Staubli VAL3: GeometryRS.dtx

public bool bIsScara = true
public bool bLinear = true
public bool bUseUserCenter
public bool bUseUserLimit = true
public num nSyncDist = 1
public num nWinDownStream
public num nWinUpStream
pointRs pVision[3]
  [0] = {x=319.933347, y=-456.969728, z=-77.119399, rx=-180, ry=0, rz=-52.793717, shoulder=lefty, fatherId=world[0]}
  [1] = {x=263.701989, y=-456.674668, z=-77.415466, rx=-180, ry=0, rz=-52.565528, shoulder=lefty, fatherId=world[0]}
  [2] = {x=319.63368, y=-491.966912, z=-77.81394, rx=-180, ry=0, rz=-52.883744, shoulder=lefty, fatherId=world[0]}
pointRs pWinCenter = {fatherId=world[0]}
pointRs pWinDown[2]
  [0] = {x=318.427982, y=-333.773146, z=-74.456462, rx=-180, ry=0, rz=-57.183953, shoulder=lefty, fatherId=world[0]}
  [1] = {x=157.577697, y=-587.439358, z=-78.679395, rx=-180, ry=0, rz=-35.162686, shoulder=lefty, fatherId=world[0]}
pointRs pWinMiddle = {fatherId=world[0]}
pointRs pWinUp[2]
  [0] = {x=690.465999, y=-334.533545, z=-72.519533, rx=180, ry=0, rz=-90.661775, shoulder=lefty, fatherId=world[0]}
  [1] = {x=529.205292, y=-587.50669, z=-76.616089, rx=-180, ry=0, rz=-72.007476, shoulder=lefty, fatherId=world[0]}
tool pointer = {z=100, fatherId=flange[0], ioLink=valve1}
